{attribute addProperty BoxType "EM3712-0000-0016"}
{attribute addProperty Id "AI_Input_ChannelAT %I*ARRAY[0..1] OF AI_Input_Channel_D7666BC26480WcStateAT %I*WcState_F855686C1620InfoDataAT %I*InfoData_BC63D37F80100"}
{attribute addProperty CRC "1915253442"}
{attribute addProperty SizeInBites "160"}
{attribute addProperty SizeInBytes "20"}
TYPE EM3712_5379163E :
STRUCT
	{attribute addProperty Name "AI_Input_Channel"}
	AI_Input_Channel : ARRAY[0..1] OF AI_Input_Channel_D7666BC2;
	{attribute addProperty Name "WcState"}
	WcState : WcState_F855686C;
	{attribute addProperty Name "InfoData"}
	InfoData : InfoData_BC63D37F;
END_STRUCT
END_TYPE

(* stored: Version 1.2.0.0, ProductVersion 3.1.4024.9
   DUT EM3712_5379163E: Id {6a4cce38-fb34-457c-b93b-3e9f00095dd2} *)
